INTERFACE I_Lens


PROPERTY Energy : LREAL
GET
END_GET
SET
END_SET
END_PROPERTY


PROPERTY Error : BOOL
GET
END_GET
END_PROPERTY


PROPERTY ErrorMsg : T_MaxString
GET
END_GET
END_PROPERTY

PROPERTY f1 : LREAL
GET
END_GET
END_PROPERTY


PROPERTY FocalLength : LREAL
GET
END_GET
END_PROPERTY


METHOD GetDelta : LREAL
VAR_INPUT
    fEnergy : LREAL;
    iXRayDelta : I_XRayDelta;
END_VAR
END_METHOD


PROPERTY Material : FB_Element
GET
END_GET
SET
END_SET
END_PROPERTY


PROPERTY Multiplier : INT
GET
END_GET
SET
END_SET
END_PROPERTY


PROPERTY Radius : LREAL
GET
END_GET
SET
END_SET
END_PROPERTY


METHOD SetState
VAR_INPUT
    fEnergy : LREAL;
    fRadius : LREAL;
    nMultiplier : INT;
    fbMaterial : FB_Element;
END_VAR
END_METHOD

END_INTERFACE

(* stored: Version 1.1.0.1, ProductVersion 3.1.4022.18
   Itf I_Lens: Id {8380e7cd-8922-468c-9bc8-67049010ef1b}
   Property Energy: Id {363904a5-e3f0-4d05-840c-a1a4eea03772}
   Get Get: Id {12514455-67ce-44ce-89f9-5a1b59eb39d1}
   Set Set: Id {30352178-f3bf-4986-b707-c27b0ad40194}
   Property Error: Id {7bf51103-b979-496d-a3f6-1a9fc6069fda}
   Get Get: Id {cf41a3e8-5659-4516-b4de-3112e1673a71}
   Property ErrorMsg: Id {2a2709c5-8e6f-4670-8b1e-c06b2fe7f1a9}
   Get Get: Id {0a46fe72-2275-473e-9ddd-f1e0d114aa9f}
   Property f1: Id {07193fcb-87f8-4ac9-b55d-034dbde78b6c}
   Get Get: Id {15e6b669-0015-4df7-a47a-ca1de16a908f}
   Property FocalLength: Id {fee325c2-3756-4383-a2b6-19ae22a67410}
   Get Get: Id {b5b301a0-8c4d-4387-9a91-47772da2143d}
   Method GetDelta: Id {18585902-8c14-4103-b71c-d60957054793}
   Property Material: Id {f24ca67e-b634-4d08-be9b-c1a2488c5d17}
   Get Get: Id {00afacb3-7434-4c19-894e-3762b24321b0}
   Set Set: Id {4c543551-0218-4739-a88a-851ad21005e8}
   Property Multiplier: Id {133e4a1d-9481-49a5-b4df-eb3676683970}
   Get Get: Id {cfc4bdd1-0628-4d12-ba7e-8ef94be7e3f0}
   Set Set: Id {e40f3da7-32b7-402b-a8d2-1dca20c55b83}
   Property Radius: Id {b4d4c109-16a7-40ac-aa76-972f60c274fd}
   Get Get: Id {241741a0-f5ed-4b0f-bb0a-9d9a105efca3}
   Set Set: Id {a4c344ef-5646-4cb5-a27d-f6d1d2e14660}
   Method SetState: Id {49ceaaa0-7087-47f6-bee4-9d13df8293ff} *)
